// SIMATIC S7-200 project (STEP 7-Micro/WIN), CPU 224XP CN REL 02.01

ORGANIZATION_BLOCK MAIN:OB1
TITLE=PROGRAM COMMENTS
BEGIN
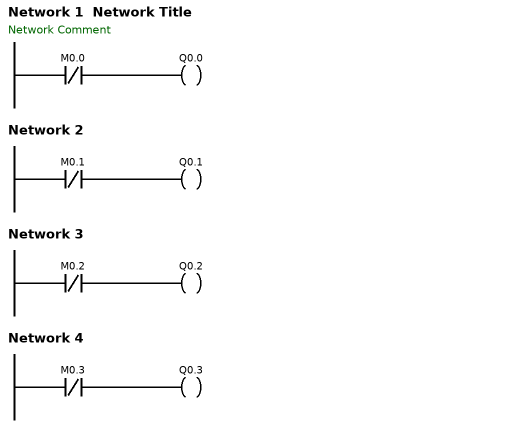
Network 1 // Network Title
// Network Comment
LDN    M0.0
=      Q0.0
Network 2
LDN    M0.1
=      Q0.1
Network 3
LDN    M0.2
=      Q0.2
Network 4
LDN    M0.3
=      Q0.3
END_ORGANIZATION_BLOCK
